FUNCTION_BLOCK FB_Obj_AddParam EXTENDS FB_BA_View
VAR
	TestAVal			: FB_UDef_AVal				:= (iParent:=THIS^,		sDescription:='My user defined analog object',				eMode:=E_UDef_Mode.eAdd);
	TestAValEx			: FB_UDef_AValEx			:= (iParent:=THIS^,		sDescription:='Another user defined enabled analog object',	eMode:=E_UDef_Mode.eSubstract);
END_VAR
VAR
	{region 'Test'}
		nOffset			: UINT						:= 3;
	{endregion}
END_VAR

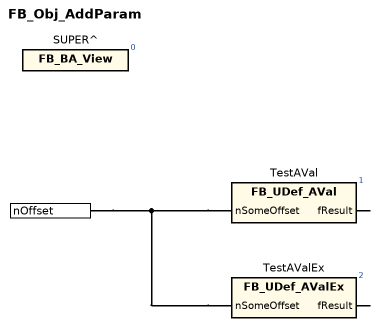
SUPER^(); // FB_BA_View
TestAVal(nSomeOffset := nOffset); // FB_UDef_AVal
TestAValEx(nSomeOffset := nOffset); // FB_UDef_AValEx

END_FUNCTION_BLOCK

(* stored: Version 1.1.0.1, ProductVersion 3.1.4024.11
   POU FB_Obj_AddParam: Id {ee9c847e-86ab-4ab1-a8c8-e6dfc4e4d446}, SpecialFunc None *)
